TYPE IM2Glue :  //备胶方法st
STRUCT
    Start1:BOOL;   //备胶启动
	Done1:BOOL;   //备胶完成
	bActioning:BOOL;//备胶动作中	
	bAction2ing:BOOL;//贴胶动作中	

	Start2:BOOL;   //贴胶启
	iTagetPos : INT;  //贴胶位置
    Done2:BOOL;  //贴胶动作完成
	

	Reset:BOOL;  //复位
	AutoRuning:BOOL;  //运行中信号

END_STRUCT
END_TYPE

(* stored: Version 1.1.0.1, ProductVersion 3.1.4024.9
   DUT IM2Glue: Id {742edbe2-70b7-49b7-9cf4-6ec92cf6c7b1} *)
